Staubli VAL3: scan_bestFit.pgx

program scan_bestFit(tool x_tTool, num x_nIndex, point& x_pBestFit[])
  local num i
  local bool l_bPrevious
  local bool l_bNext
  local point l_pCheck
  local point l_pHere
  local num l_nSize
  local num l_nDistanceNext
  local num l_nDistancePrev
  local num l_nStopPrev
  local num l_nStopNext
  local num i_from
  local num i_to
  local bool l_bOk
  local num l_nMoveType
  local joint l_jResult
  local joint l_jJoint[3]
begin
  // save the point
  // pBestFit [0] -> previous
  // pBestFit [1] -> actual
  // pBestFit [2] -> next
  // scan all
  call getSizeItem(true,l_nSize)
  l_nDistanceNext=10000
  l_nDistancePrev=10000
  call getMoveType(l_nMoveType,x_nIndex,true)
  // search the three point
  if x_nIndex>0
    l_bPrevious=true
    call getJointData(l_jJoint[0],x_tTool,true,x_nIndex-1)
    x_tTool=flange
    pBestFit[0]=jointToPoint(x_tTool,world,l_jJoint[0])
  endIf
  if x_nIndex<l_nSize-1 and l_nSize>1
    l_bNext=true
    call getJointData(l_jJoint[2],x_tTool,true,x_nIndex+1)
    pBestFit[2]=jointToPoint(x_tTool,world,l_jJoint[2])
  endIf
  call getJointData(l_jJoint[1],x_tTool,true,x_nIndex)
  pBestFit[1]=jointToPoint(x_tTool,world,l_jJoint[1])
  // look if the next point if is better
  if l_bNext
    if setFrame(pBestFit[1],pBestFit[2],pNull,fFrame)==0
      pCheck=here(x_tTool,fFrame)
      if pCheck.trsf.x>=0
        // scan it
        l_pCheck=pBestFit[1]
        l_pHere=here(x_tTool,world)
        // check the nearest point
        for i=0 to 0.4 step 0.1
          if l_nMoveType==0
            call interpolateJ(l_jJoint[1],l_jJoint[2],i,l_jResult,l_bOk)
            l_pCheck=jointToPoint(x_tTool,world,l_jResult)
          else
            l_pCheck.trsf=interpolateL(pBestFit[1].trsf,pBestFit[2].trsf,i)
            l_bOk=true
          endIf
          if l_nDistanceNext>=distance(l_pCheck,l_pHere) and l_bOk
            l_nDistanceNext=distance(l_pCheck,l_pHere)
            //save the value
            l_nStopNext=i
          endIf
        endFor
        // closer search
        i_from=(max(l_nStopNext-0.05,0))
        i_to=(min(l_nStopNext+0.05,1))
        for i=i_from to i_to step 0.01
          if l_nMoveType==0
            call interpolateJ(l_jJoint[1],l_jJoint[2],i,l_jResult,l_bOk)
            l_pCheck=jointToPoint(x_tTool,world,l_jResult)
          else
            l_pCheck.trsf=interpolateL(pBestFit[1].trsf,pBestFit[2].trsf,i)
            l_bOk=true
          endIf
          if l_nDistanceNext>=distance(l_pCheck,l_pHere) and l_bOk
            l_nDistanceNext=distance(l_pCheck,l_pHere)
            //save the value
            l_nStopNext=i
          endIf
        endFor
      endIf
    endIf
  endIf
  // look if there is a previous point
  if l_bPrevious
    if setFrame(pBestFit[0],pBestFit[1],pNull,fFrame)==0
      pCheck=here(x_tTool,fFrame)
      // scan it
      if pCheck.trsf.x>=0
        // scan it
        l_pCheck=pBestFit[1]
        l_pHere=here(x_tTool,world)
        // check the nearest point
        for i=0.6 to 1 step 0.1
          if l_nMoveType==0
            call interpolateJ(l_jJoint[0],l_jJoint[1],i,l_jResult,l_bOk)
            l_pCheck=jointToPoint(x_tTool,world,l_jResult)
          else
            l_pCheck.trsf=interpolateL(pBestFit[0].trsf,pBestFit[1].trsf,i)
            l_bOk=true
          endIf
          if l_nDistancePrev>=distance(l_pCheck,l_pHere)
            l_nDistancePrev=distance(l_pCheck,l_pHere)
            //save the value
            l_nStopPrev=i
          endIf
        endFor
        // closer search
        i_from=(max(l_nStopPrev-0.05,0))
        i_to=(min(l_nStopPrev+0.05,1))
        for i=i_from to i_to step 0.01
          if l_nMoveType==0
            call interpolateJ(l_jJoint[0],l_jJoint[1],i,l_jResult,l_bOk)
            l_pCheck=jointToPoint(x_tTool,world,l_jResult)
          else
            l_pCheck.trsf=interpolateL(pBestFit[0].trsf,pBestFit[1].trsf,i)
            l_bOk=true
          endIf
          if l_nDistancePrev>=distance(l_pCheck,l_pHere)
            l_nDistancePrev=distance(l_pCheck,l_pHere)
            //save the value
            l_nStopPrev=i
          endIf
        endFor
      endIf
    endIf
  endIf
  // go to an approach POINT
  if l_nStopNext!=0 or l_nStopPrev!=0
    if l_nDistanceNext<l_nDistancePrev
      if l_nMoveType==0
        call interpolateJ(l_jJoint[1],l_jJoint[2],l_nStopNext,l_jResult,l_bOk)
        l_pCheck=jointToPoint(x_tTool,world,l_jResult)
      else
        l_pCheck.trsf=interpolateL(pBestFit[1].trsf,pBestFit[2].trsf,l_nStopNext)
      endIf
    else
      if l_nMoveType==0
        call interpolateJ(l_jJoint[0],l_jJoint[1],l_nStopPrev,l_jResult,l_bOk)
        l_pCheck=jointToPoint(x_tTool,world,l_jResult)
      else
        ? l_nStopPrev
        l_pCheck.trsf=interpolateL(pBestFit[0].trsf,pBestFit[1].trsf,l_nStopPrev)
      endIf
    endIf
    // save it
    x_pBestFit=l_pCheck
  else
    // return the default
    x_pBestFit=pBestFit[1]
  endIf
end
